Staubli VAL3: getStrDate.pgx

program getStrDate(string x_sText (dimensions=1), string& x_sDate[] (dimensions=1))
begin
  //获取point,joint和速度值
  call split(x_sText,"/",x_sDate)
end
